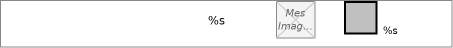
VISUALIZATION VISU_LIGNE_EAU_No_VE  // 453x48
VAR_IN_OUT
	m_Input_LIGNE_EAU : BLOCK_LIGNE_REF;
END_VAR
    Polyline (451,20)
    Polyline (80,20)
    Polyline (129,20)
    Polygon (140,20)
    Polygon (317,20)
    Rectangle (380,15 65x31), "%s", text variable: m_Input_LIGNE_EAU.mnemo_DEX, invisible if: m_Input_LIGNE_EAU.CONF_NO_DexT
    Rectangle (344,1 33x33), colour toggle: (m_Input_LIGNE_EAU.IN_DExT) <> 0, invisible if: (m_Input_LIGNE_EAU.CONF_NO_DexT) <> 0
    Polyline (16,8)
    Polyline (24,15)
    Rectangle (154,5 125x31), "%s", text variable: m_Input_LIGNE_EAU.mnemo
    Image (276,1 39x37), invisible if: NOT m_Input_LIGNE_EAU.STATE_NOK, image: MesImages.warning
END_VISUALIZATION

(* stored: Version 1.1.0.1, ProductVersion 3.1.4024.10
   Visu VISU_LIGNE_EAU_No_VE: Id {af491c4b-1cd1-42c8-8121-2faeae61f6cf} *)
